// TIA Portal V19 export
TYPE "OB82_vars"
TITLE = Variable structure of OB82 Diagnostic Interrupt
   STRUCT
      IO_State { ExternalAccessible := 'False'; ExternalVisible := 'False'; ExternalWritable := 'False'} : Word;   // IO state of the HW object
      LADDR { ExternalAccessible := 'False'; ExternalVisible := 'False'; ExternalWritable := 'False'} : HW_ANY;   // Hardware identifier
      Channel { ExternalAccessible := 'False'; ExternalVisible := 'False'; ExternalWritable := 'False'} : UInt;   // Channel number
      MultiError { ExternalAccessible := 'False'; ExternalVisible := 'False'; ExternalWritable := 'False'} : Bool;   // =true if more than one error is present
   END_STRUCT;
END_TYPE
